Universal Robots PolyScope program: Tall_PHomeToInvC.urp

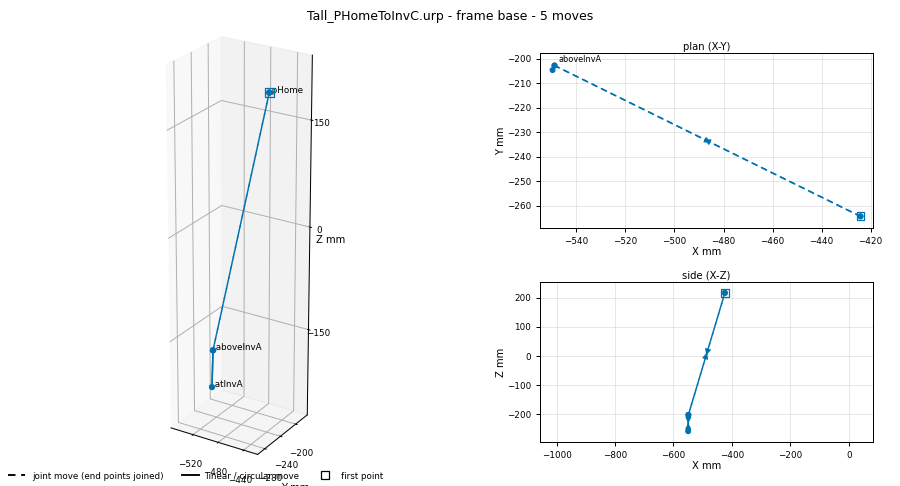
[picture p0: tool path of Tall_PHomeToInvC.urp in frame base, 5 of 5 moves have a stored position in this frame; points joined in program order, loops and branches not executed]
Program Tall_PHomeToInvC (installation=admin directory=/programs/THU_530PM/Final createdIn=3.8.0.61336 lastSavedIn=3.15.8.106339 robotSerialNumber=2015350925)
Calibrated DH parameters: a=[0, -0.425, -0.39225, 0, 0, 0]; d=[0.089159, 0, 0, 0.10915, 0.09465, 0.0823]; alpha=[1.570796, 0, 0, 1.570796, -1.570796, 0]; deltaTheta=[0, 0, 0, 0, 0, 0]
Robot Program (runOnlyOnce=true)
  Set DigitalOutput pin=digital_out[0]; digitalValue=1
  Wait Sleep waitTime=1
  Call _adminLinearIndex3
  Wait Sleep waitTime=1
  MoveJ speed 180 deg/s, acceleration 100 deg/s^2 (useActiveTCP=true)
    Waypoint pHome: TCP in base x=-424.177 y=-264.287 z=215.871 mm, rx=-1.1973 ry=-2.8917 rz=-0.0084 rad; joints [224.995, -90.007, -90.004, -90.013, 89.257, -0.019] deg; flange x=-422.26 y=-266.331 z=431.752 mm, rx=-1.1973 ry=-2.8917 rz=-0.0084 rad
    Waypoint aboveInvA: TCP in base x=-548.91 y=-202.799 z=-201.342 mm, rx=-1.2068 ry=2.899 rz=-0.0022 rad; joints [210.98, -128.201, -108.055, -33.815, 90.09, -104.223] deg; flange x=-549.316 y=-202.646 z=14.558 mm, rx=-1.2068 ry=2.899 rz=-0.0022 rad
  MoveL speed 250 mm/s, acceleration 500 mm/s^2 (useActiveTCP=true) feature=Base
    Waypoint atInvA: TCP in base x=-549.712 y=-204.656 z=-257.326 mm, rx=-1.2069 ry=2.8991 rz=-0.0022 rad; joints [211.098, -135.126, -107.409, -27.526, 90.089, -104.106] deg; flange x=-550.085 y=-204.489 z=-41.426 mm, rx=-1.2069 ry=2.8991 rz=-0.0022 rad
    Set DigitalOutput pin=digital_out[0]; digitalValue=0
    Wait Sleep waitTime=1
    Waypoint aboveInvA: motionParameters(blendRadius=0.01); TCP in base x=-548.91 y=-202.799 z=-201.342 mm, rx=-1.2068 ry=2.899 rz=-0.0022 rad; joints [210.98, -128.201, -108.055, -33.815, 90.09, -104.223] deg; flange x=-549.316 y=-202.646 z=14.558 mm, rx=-1.2068 ry=2.899 rz=-0.0022 rad
  MoveJ speed 180 deg/s, acceleration 100 deg/s^2 (useActiveTCP=true)
    Waypoint pHome: TCP in base x=-424.177 y=-264.287 z=215.871 mm, rx=-1.1973 ry=-2.8917 rz=-0.0084 rad; joints [224.995, -90.007, -90.004, -90.013, 89.257, -0.019] deg; flange x=-422.26 y=-266.331 z=431.752 mm, rx=-1.1973 ry=-2.8917 rz=-0.0084 rad
SubProgram -> _adminLinearIndex3
SubProgram _adminLinearIndex3 (keepSynchronizedWithDisk=false) programFile=/programs/me345_admin/_adminLinearIndex3.urp
  Folder Move_linear_slide_Index3
    var_1 := False
    Loop While (checkContinuously=false) expression=var_1≟ False
      var_1 := socket_open("10.241.34.48",4001)
    var_3 := 1
    Send := "s r0x24 21"
    Script: socket_send_string(Send)
    Script: socket_send_byte(13)
    Send_Reply := socket_read_string()
    Send := "s r0xca 112778"
    Script: socket_send_string(Send)
    Script: socket_send_byte(13)
    Send_Reply := socket_read_string()
    Send := "t 1"
    Script: socket_send_string(Send)
    Script: socket_send_byte(13)
    Send_Reply := socket_read_string()
    Loop While (checkContinuously=false) expression=var_3≠0
      Send := "g r0xA0"
      Script: socket_send_string(Send)
      Script: socket_send_byte(13)
      var_3 := socket_get_var("v")
      Wait Sleep waitTime=0.1
    Script: socket_close()
    Script: sync()
